FUNCTION SinusFunction : REAL
VAR_INPUT
	A : REAL;
	yOffset : REAL;
	w : REAL;
	t : REAL;
END_VAR
VAR
END_VAR

SinusFunction := A * SIN(w*t) + yOffset;

END_FUNCTION

(* stored: Version 1.1.0.1, ProductVersion 3.1.4022.10
   POU SinusFunction: Id {e59db478-07c7-4fb1-a0f8-5383e0b8798e}, SpecialFunc None *)
